{attribute 'GeneratedUsingTerminal: EPP4174-0002-0016'}
{attribute addProperty BoxType "EPP4174-0002-0016"}
{attribute addProperty Id "Analog_outputAT %Q*INT2"}
{attribute addProperty CRC "3128867708"}
{attribute addProperty Size "2"}
TYPE AO_Outputs_Channel_BA7EBB7C :
STRUCT
	{attribute addProperty Name "Analog_output"}
	Analog_output AT %Q* : INT;
END_STRUCT
END_TYPE

(* stored: Version 1.2.0.0, ProductVersion 3.1.4024.9
   DUT AO_Outputs_Channel_BA7EBB7C: Id {ad946fa4-8502-49ee-80fa-ad68e59f7990} *)
